// TIA Portal project "factoryio test" (V19)

(* hardware
DEVICE "S71500/ET200MP-Station_1"  S7-1500 station
   slot 0: "Profilschiene_0"  6ES7 590-1***0-0AA0
   slot 1: "PLC_1"  CPU 1511-1 PN  6ES7 511-1AK00-0AB0  V1.8
   slot 2: "AI 8xU/I/RTD/TC ST_1"  AI 8xU/I/RTD/TC ST  6ES7 531-7KF00-0AB0  V2.0
   slot 3: "AI 8xU/I/RTD/TC ST_2"  AI 8xU/I/RTD/TC ST  6ES7 531-7KF00-0AB0  V2.0
   slot 4: "AI 8xU/I/RTD/TC ST_3"  AI 8xU/I/RTD/TC ST  6ES7 531-7KF00-0AB0  V2.0
   slot 5: "AI 8xU/I/RTD/TC ST_4"  AI 8xU/I/RTD/TC ST  6ES7 531-7KF00-0AB0  V2.0
   slot 6: "DI 16x24VDC BA_1"  DI 16x24VDC BA  6ES7 521-1BH10-0AA0  V1.0
*)

// ===== PLC "PLC_1"  CPU 1511-1 PN =====

VAR_GLOBAL   // PLC tag table "Standard-Variablentabelle"
   "Tag_1" AT %E0.0 : Bool;
   "Tag_2" AT %A0.0 : Bool;
   "Tag_3" AT %E0.1 : Bool;
END_VAR

VAR_GLOBAL   // PLC tag table "control panel"
   "start button" AT %I0.0 : Bool;
   "reset button" AT %I0.1 : Bool;
   "stop button" AT %I0.2 : Bool;
   "emergency stop" AT %I0.3 : Bool;
   "start button light" AT %Q0.0 : Bool;
   "reset button light" AT %Q0.1 : Bool;
   "stop button light" AT %Q0.2 : Bool;
   "system start" AT %Q0.3 : Bool;
   "system fault" AT %Q0.4 : Bool;
   "system stop" AT %Q0.5 : Bool;
END_VAR

VAR_GLOBAL   // PLC tag table "conveyor 0"
   "motor +" AT %Q3.7 : Bool;
   "motor -" AT %Q3.6 : Bool;
   "encoder A" AT %I2.7 : Bool;
   "encoder B" AT %I2.6 : Bool;
   "sensor" AT %I3.7 : Bool;
END_VAR

VAR_GLOBAL   // PLC tag table "conveyor 1"
   "motor +(1)" AT %Q3.5 : Bool;
   "motor -(1)" AT %Q3.4 : Bool;
   "encoder A(1)" AT %I2.5 : Bool;
   "encoder B(1)" AT %I2.4 : Bool;
   "sensor(1)" AT %I3.6 : Bool;
END_VAR

VAR_GLOBAL   // PLC tag table "conveyor 2"
   "motor +(2)" AT %Q3.3 : Bool;
   "motor -(2)" AT %Q3.2 : Bool;
   "encoder A(2)" AT %I2.2 : Bool;
   "encoder B(2)" AT %I2.3 : Bool;
   "sensor(2)" AT %I3.5 : Bool;
END_VAR

DATA_BLOCK "conveyor 2"   // DB3
{ S7_Optimized_Access := 'TRUE' }
VERSION : 0.1
// stored: InstanceOfName conveyor
"conveyor"
BEGIN
END_DATA_BLOCK

DATA_BLOCK "conveyor 0"   // DB5
{ S7_Optimized_Access := 'TRUE' }
VERSION : 0.1
// stored: InstanceOfName conveyor
"conveyor"
BEGIN
END_DATA_BLOCK

DATA_BLOCK "conveyor 1"   // DB6
{ S7_Optimized_Access := 'TRUE' }
VERSION : 0.1
// stored: InstanceOfName conveyor
"conveyor"
BEGIN
END_DATA_BLOCK

FUNCTION_BLOCK "conveyor"   // FB1, LAD
{ S7_Optimized_Access := 'TRUE' }
VERSION : 0.1
   VAR_INPUT
      enable : Bool;
      "encoder A" : Bool;
      "encoder B" : Bool;
   END_VAR
   VAR_OUTPUT
      "running feedback" : Bool;
      "motor +" : Bool;
      "motor -" : Bool;
   END_VAR
   VAR
      IEC_Timer_0_Instance : TOF_TIME;
      IEC_Timer_0_Instance_1 : TOF_TIME;
   END_VAR
BEGIN

REGION Network 1
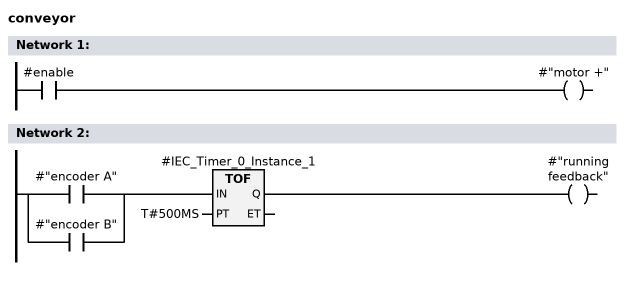
   RUNG wire#powerrail
      Contact( #enable )
      Coil( #"motor +" )
   END_RUNG
   // the same network as SCL:
   #"motor +" := #enable;
END_REGION

REGION Network 2
   #IEC_Timer_0_Instance_1(IN := #"encoder A" OR #"encoder B", PT := T#500MS);   // TOF
   #"running feedback" := #IEC_Timer_0_Instance_1.Q;
END_REGION
END_FUNCTION_BLOCK

FUNCTION "MHJ-PLC-Lab-Function-S71500" : Void   // FC9000, SCL
{ S7_Optimized_Access := 'TRUE' }
VERSION : 0.1
   VAR_TEMP
      Value : Byte;
      ForCounter : Int;
   END_VAR
   VAR CONSTANT
      Value_01_DW : DWord := 16#1223_5486;
      Value_02_DW : DWord := 16#A6C9_D1F5;
   END_VAR
BEGIN

   #Value:=PEEK(area := 16#82,
        dbNumber := 0,
        byteOffset := 511);
   #Value := #Value + 1;

   POKE(area := 16#82,
        dbNumber := 0,
        byteOffset := 511,
        value := #Value);

   POKE(area := 16#82,
        dbNumber := 0,
        byteOffset := 1016,
        value := #Value_01_DW);
   POKE(area := 16#82,
        dbNumber := 0,
        byteOffset := 1020,
        value := #Value_02_DW);

   FOR #ForCounter := 0 TO 63 DO
       #Value:=PEEK(area := 16#1,
            dbNumber := 0,
            byteOffset := #ForCounter);
       POKE(area := 16#81,
            dbNumber := 0,
            byteOffset := #ForCounter,
            value := #Value);
   END_FOR;
   #Value := PEEK(area := 16#1,
                  dbNumber := 0,
                  byteOffset := 512);
   POKE(area := 16#82,
        dbNumber := 0,
        byteOffset := 512,
        value := #Value);
END_FUNCTION

ORGANIZATION_BLOCK "Main"   // OB1, LAD, ProgramCycle
TITLE = "Main Program Sweep (Cycle)"
{ S7_Optimized_Access := 'TRUE' }
VERSION : 0.1
   VAR_INPUT
      Initial_Call : Bool;   // Initial call of this OB
      Remanence : Bool;   // =True, if remanent data are available
   END_VAR
   VAR_TEMP
      "start 1" : Bool;
      "start 2" : Bool;
      "motor 0 enable" : Bool;
      "motor 0 feedback" : Bool;
      "sensor 0 feedback" : Bool;
      "motor 1 enable" : Bool;
      "motor 1 feedback" : Bool;
      "sensor 1 feedback" : Bool;
      "motor 2 enable" : Bool;
      "motor 2 feedback" : Bool;
      "sensor 2 feedback" : Bool;
      Constant : Bool;
   END_VAR
   VAR CONSTANT
      "conveyor clear time" : Bool;
   END_VAR
BEGIN

REGION Network 1
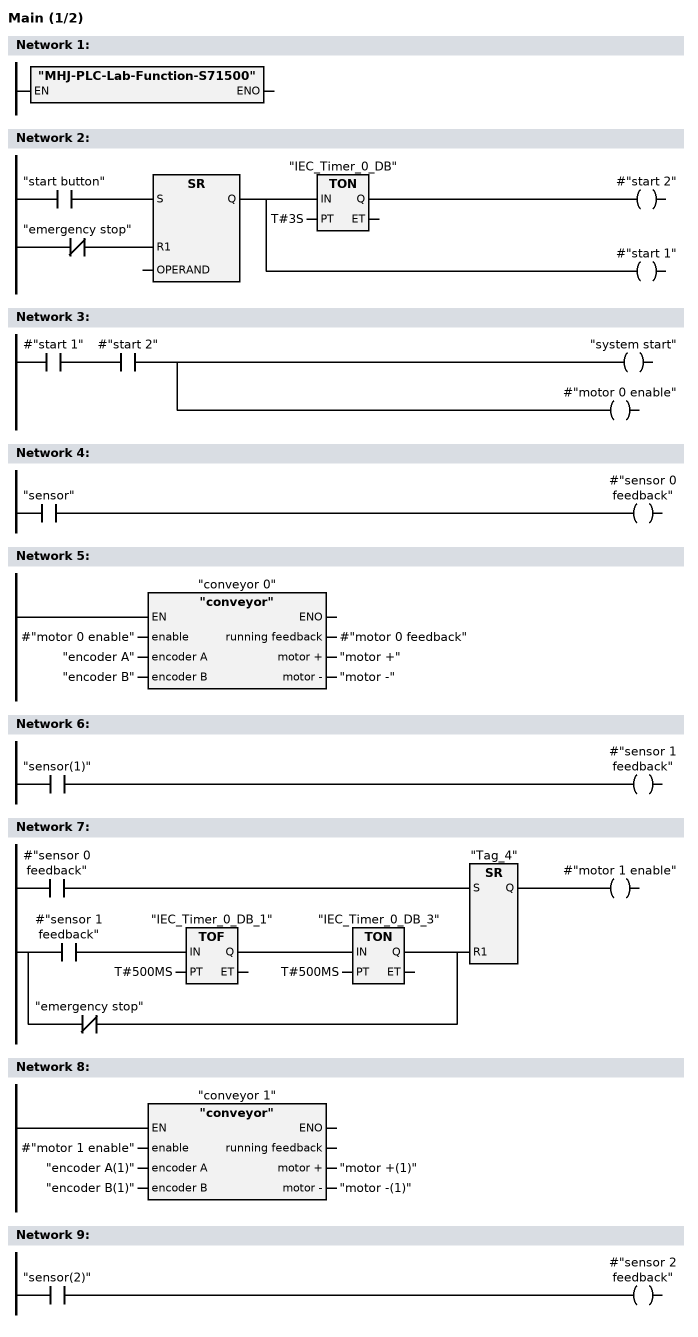
   RUNG wire#powerrail
      "MHJ-PLC-Lab-Function-S71500"()
   END_RUNG
   // the same network as SCL:
   "MHJ-PLC-Lab-Function-S71500"();
END_REGION

REGION Network 2
   IF "start button" THEN
       <??.?> := TRUE;   // SR flip-flop
   END_IF;
   IF NOT "emergency stop" THEN <??.?> := FALSE; END_IF;
   "IEC_Timer_0_DB".TON(IN := <??.?>, PT := T#3S);
   #"start 2" := "IEC_Timer_0_DB".Q;
   #"start 1" := <??.?>;
END_REGION

REGION Network 3
   RUNG wire#powerrail
      Contact( #"start 1" )
      Contact( #"start 2" )
      wire#w1
      Coil( "system start" )
   END_RUNG
   RUNG wire#w1
      Coil( #"motor 0 enable" )
   END_RUNG
   // the same network as SCL:
   "system start" := #"start 1" AND #"start 2";
   #"motor 0 enable" := "system start";
END_REGION

REGION Network 4
   RUNG wire#powerrail
      Contact( "sensor" )
      Coil( #"sensor 0 feedback" )
   END_RUNG
   // the same network as SCL:
   #"sensor 0 feedback" := "sensor";
END_REGION

REGION Network 5
   RUNG wire#powerrail
      "conveyor 0"(enable := #"motor 0 enable", "encoder A" := "encoder A", "encoder B" := "encoder B", "running feedback" => #"motor 0 feedback", "motor +" => "motor +", "motor -" => "motor -")
   END_RUNG
   // the same network as SCL:
   "conveyor 0"(enable := #"motor 0 enable",   // "conveyor"
                "encoder A" := "encoder A",
                "encoder B" := "encoder B",
                "running feedback" => #"motor 0 feedback",
                "motor +" => "motor +",
                "motor -" => "motor -");
END_REGION

REGION Network 6
   RUNG wire#powerrail
      Contact( "sensor(1)" )
      Coil( #"sensor 1 feedback" )
   END_RUNG
   // the same network as SCL:
   #"sensor 1 feedback" := "sensor(1)";
END_REGION

REGION Network 7
   "IEC_Timer_0_DB_1".TOF(IN := #"sensor 1 feedback", PT := T#500MS);
   "IEC_Timer_0_DB_3".TON(IN := "IEC_Timer_0_DB_1".Q, PT := T#500MS);
   IF #"sensor 0 feedback" THEN
       "Tag_4" := TRUE;   // SR flip-flop
   END_IF;
   IF "IEC_Timer_0_DB_3".Q OR NOT "emergency stop" THEN "Tag_4" := FALSE; END_IF;
   #"motor 1 enable" := "Tag_4";
END_REGION

REGION Network 8
   RUNG wire#powerrail
      "conveyor 1"(enable := #"motor 1 enable", "encoder A" := "encoder A(1)", "encoder B" := "encoder B(1)", "running feedback" =>, "motor +" => "motor +(1)", "motor -" => "motor -(1)")
   END_RUNG
   // the same network as SCL:
   "conveyor 1"(enable := #"motor 1 enable",   // "conveyor"
                "encoder A" := "encoder A(1)",
                "encoder B" := "encoder B(1)",
                "motor +" => "motor +(1)",
                "motor -" => "motor -(1)");
END_REGION

REGION Network 9
   RUNG wire#powerrail
      Contact( "sensor(2)" )
      Coil( #"sensor 2 feedback" )
   END_RUNG
   // the same network as SCL:
   #"sensor 2 feedback" := "sensor(2)";
END_REGION

REGION Network 10
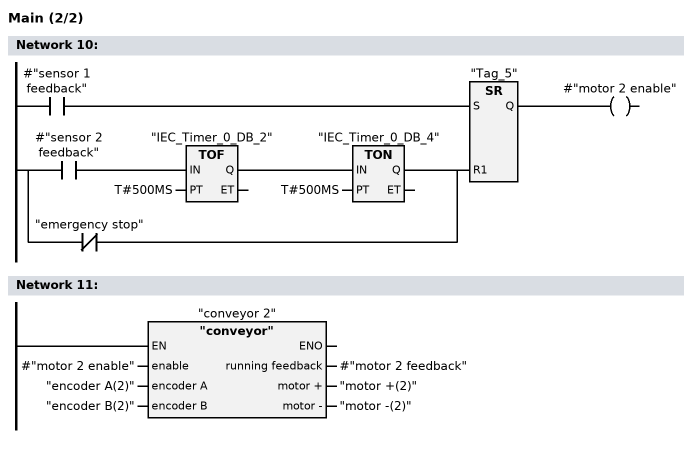
   "IEC_Timer_0_DB_2".TOF(IN := #"sensor 2 feedback", PT := T#500MS);
   "IEC_Timer_0_DB_4".TON(IN := "IEC_Timer_0_DB_2".Q, PT := T#500MS);
   IF #"sensor 1 feedback" THEN
       "Tag_5" := TRUE;   // SR flip-flop
   END_IF;
   IF "IEC_Timer_0_DB_4".Q OR NOT "emergency stop" THEN "Tag_5" := FALSE; END_IF;
   #"motor 2 enable" := "Tag_5";
END_REGION

REGION Network 11
   RUNG wire#powerrail
      "conveyor 2"(enable := #"motor 2 enable", "encoder A" := "encoder A(2)", "encoder B" := "encoder B(2)", "running feedback" => #"motor 2 feedback", "motor +" => "motor +(2)", "motor -" => "motor -(2)")
   END_RUNG
   // the same network as SCL:
   "conveyor 2"(enable := #"motor 2 enable",   // "conveyor"
                "encoder A" := "encoder A(2)",
                "encoder B" := "encoder B(2)",
                "running feedback" => #"motor 2 feedback",
                "motor +" => "motor +(2)",
                "motor -" => "motor -(2)");
END_REGION
END_ORGANIZATION_BLOCK